# B&R Automation Studio project CoffeeMachine
Automation Studio 4.2.3.159; Default project

## Configuration Simulation

CPU , AutomationRuntime H4.23, Build 4.1.2

### Task classes (Cpu.sw)
```
Cyclic#1 (cycle 100000 us, tolerance 10000000 us):
  Program <- Program.prg
Cyclic#4 (cycle 1000000 us, tolerance 10000000 us):
  program1 <- Program.prg
Libraries: AsIecCon, astime
```

### Hardware
```
PC_any : PC_any v1.1.0.0 (OrderNumber=PC)
  ConfigurationID = CoffeeMachine_Simulation
  Cyclic1Duration = 100000
  Cyclic1Tolerance = 10000000
  Cyclic2Duration = 200000
  Cyclic2Tolerance = 10000000
  Cyclic3Duration = 500000
  Cyclic3Tolerance = 10000000
  Cyclic4Duration = 1000000
  Cyclic4Tolerance = 10000000
  Cyclic5Duration = 2000000
  Cyclic5Tolerance = 10000000
  Cyclic6Duration = 3000000
  Cyclic6Tolerance = 12000000
  Cyclic7Duration = 4000000
  Cyclic7Tolerance = 12000000
  Cyclic8Duration = 5000000
  Cyclic8Tolerance = 30000000
```

## Logical view

Binary libraries used (declarations not repeated): Runtime, Operator, AsIecCon, astime


### Program Logical/Program (ANSIC)

#### Cyclic.cpp - Cyclic code
```cpp
#include <bur/plctypes.h>
#ifdef _DEFAULT_INCLUDES
	#include <AsDefault.h>
#endif

#include "class_dec.h"
#include "auxiliary.h"

myRobot robot;

void _CYCLIC ProgramCyclic(void)
{
	Input();
	robot.Operation();
}
```

#### auxiliary.h
```c
#ifndef __AUXILIARY_H
#define __AUXILIARY_H

#include <iostream>
#include <string.h>

using namespace std;

/*@note
	用於存儲用戶輸入的內容
*/
typedef struct
	{
		char OperationType[11];
		char CSName[11];
		float para1;
		float para2;
		float para3;
	}InputCom;

extern InputCom input;

void Input();
float Extraction(char* str);
float Index1(int n);
float Index2(int n);

#endif
```

#### class_dec.h
```c
#ifndef __CLASS_DEC_H
#define __CLASS_DEC_H

#include <iostream>
#include <vector>
//#include <Eigen/Dense>
#include <math.h>

using namespace std;
//using Eigen::MatrixXd;

class CS
	{
		public:
			CS();
			void Set(char n[11],float a,float b,float c);
			char* GetName();
			void Insert(float a,float b);
			void Transform();
		protected:
			char name[11];
			float x;
			float y;
			float angle;
			float para1;
			float para2;
	};

class myRobot
	{
		public:
			myRobot();
			void Set(float a,float b);
			void Operation();
			void PTPMove();
			void Show();
		protected:
			float angle1;
			float angle2;
			vector<CS> cs_vector;
			vector<CS>::iterator it;
	};

extern myRobot robot;

#endif
```

#### class_def.cpp
```cpp
/*************************************************************************************************/
/*@note
	這個文件里定義了所有的類的成員函數
*/

/**includes***************************************************************************************/
#include "auxiliary.h"
#include "class_dec.h"

/**CS::Fuctions***********************************************************************************/

/*@note
	CS的構造函數
*/
CS::CS()
	{
		strcpy(name,"TCS");
		x=0;
		y=0;
		angle=0;
	}

/*@note
	用來設定新建坐標系相對於世界坐標系的平移、旋轉量
*/
void CS::Set(char n[11],float a,float b,float c)
	{
		strcpy(name,n);
		x=a;
		y=b;
		angle=c;
	}

/*@note
	獲取坐標系名稱
*/
char* CS::GetName()
	{
		return name;
	}

/*@note
	插入該坐標系下用戶要求機器人到達的坐標
*/
void CS::Insert(float a,float b)
	{
		para1=a;
		para2=b;
	}

/*@note
	將該坐標系下的坐標變換至世界坐標系并更新關節坐標系中的坐標值
*/
void CS::Transform()
{
		/*MatrixXd mov(3,3);
		mov(0,0)=cos(angle*0.0174533);
		mov(0,1)=sin(angle*0.0174533);
		mov(0,2)=x;
		mov(1,0)=-sin(angle*0.0174533);
		mov(1,1)=cos(angle*0.0174533);
		mov(1,2)=y;
		mov(2,0)=0;
		mov(2,1)=0;
		mov(2,2)=1;
		MatrixXd coor_TCS(3,1);
		coor_TCS(0,0)=para1;
		coor_TCS(1,0)=para2;
		coor_TCS(2,0)=1;
		MatrixXd coor_WCS(3,1);
		coor_WCS=mov*coor_TCS;*/

	float w_para1;
	float w_para2;
	w_para1=para1*cos(angle*0.0174533)+para2*sin(angle*0.0174533);
	w_para2=-para1*sin(angle*0.0174533)+para2*cos(angle*0.0174533);

	if((w_para1*w_para1+w_para2*w_para2)>400)    //這裡假定機器人兩個手臂的長度都是10，所以半徑20的圓以外的地方是到不了的
	{
		cout<<"Robot can't reach that point!"<<endl;
		robot.Set(90,180);
	}
	else
	{
		cout<<"The coordinates of the Robot in WCS are shown as below:"<<endl<<"("<<w_para1<<","<<w_para2<<")"<<endl;
		robot.Set((acos(sqrt(w_para1*w_para1+w_para2*w_para2)/20)+atan(w_para2/w_para1))*57.29578,\
			(2*(1.5707963-acos(sqrt(w_para1*w_para1+w_para2*w_para2)/20)))*57.29578);
	}
}

/**myRobot::Functions*****************************************************************************/

/*@note
	構造函數
*/
myRobot::myRobot()
	{
		angle1=90;
		angle2=180;
		CS* p;
		p=new CS;
		char str[4]={'W','C','S','\0'};
		p->Set(str,0,0,0);
		cs_vector.push_back(*p);
	}

/*@note
	更新關節坐標系下的坐標值
*/
void myRobot::Set(float a,float b)
	{
		angle1=a;
		angle2=b;
	}

/*@note
	判斷用戶是新建坐標系還是移動機器人
*/
void myRobot::Operation()
	{

		if(strcmp(input.OperationType,"S")==0)
			{
				CS* p;
				p=new CS;
				p->Set(input.CSName,input.para1,input.para2,input.para3);
				cs_vector.push_back(*p);
			}
		else
			{
				PTPMove();
			}
	}

/*@note
	實現坐標變換并更新關節坐標系下坐標
*/
void myRobot::PTPMove()
	{
		for(it=cs_vector.begin();it!=cs_vector.end();it++)
			{
				if(strcmp(it->GetName(),input.CSName)==0)
					{
						it->Insert(input.para1,input.para2);
						it->Transform();
						Show();
						break;
					}
			}
	}

/*@note
	顯示關節坐標系下坐標
*/
void myRobot::Show()
	{
		cout<<"The coordinates of the Robot in Joint_CS are shown as below:"<<endl<<"("<<angle1<<","<<angle2<<")"<<endl;
	}
```

#### auxiliary.cpp
```cpp
#include "auxiliary.h"

InputCom input;

void Input()
	{
		char str[11];
		cout<<"Input OperationType 'S'or'M':"<<endl;
		cin>>str;
		strcpy(input.OperationType,str);
		cout<<"Input CSName:"<<endl;
		cin>>str;
		strcpy(input.CSName,str);
		cout<<"Input para1:"<<endl;
		cin>>str;
		input.para1=Extraction(str);
		cout<<"Input para2:"<<endl;
		cin>>str;
		input.para2=Extraction(str);
		if(strcmp(input.OperationType,"S")==0)
			{
				cout<<"Input para3:"<<endl;
				cin>>str;
				input.para3=Extraction(str);
			}
		else
			{
				input.para3=0;
			}
	}

float Extraction(char* str)
	{
		int i,k;
		float a=0;
		for(i=0;str[i]!='\0';i++)
			{
				if(str[i]=='.')
					{
						k=i;
					}
			}
		if(str[0]=='-')
			{
				for(i=0;i<k-1;i++)
					{
						a+=((float)str[k-i-1]-48)*Index1(i);
					}
				for(i=1;str[k+i]!='\0';i++)
					{
						a+=((float)str[k+i]-48)*Index2(i);
					}
				a=-a;
			}
		else
			{
				for(i=0;i<k;i++)
					{
						a+=((float)str[k-i-1]-48)*Index1(i);
					}
				for(i=1;str[k+i]!='\0';i++)
					{
						a+=((float)str[k+i]-48)*Index2(i);
					}
			}
		return a;
	}

float Index1(int n)
	{
		float a=1,i;
		for(i=n;i!=0;i--)
			{
				a*=10;
			}
		return a;
	}

float Index2(int n)
	{
		float a=1,i;
		for(i=n;i!=0;i--)
			{
				a*=0.1;
			}
		return a;
	}
```

Listed in the project but not available here: Logical/Global.typ, Logical/Program/Init.cpp, Logical/Program/Exit.cpp, Logical/Program/Types.typ, Logical/Program/Variables.var
